FUNCTION_BLOCK T_AdsWrite EXTENDS T_NamedBase IMPLEMENTS I_TaskState;
VAR
   _readWriteOpts : ST_AdsReadWriteOptions;

   write : ADSWRITE;
   {attribute 'to_String'}
   state, prevState : (
      IDLE,
      REQUEST,
      WAIT_FOR_RESPONSE,
      DONE_STATE,
      ERROR_STATE
   );

   lastErrorId : UDINT;

END_VAR
VAR CONSTANT
   NO_ERR : UDINT := 0;
   LOG_DEBUG : DWORD := 0;
   LOG_INFO : DWORD := ADSLOG_MSGTYPE_HINT;
   LOG_WARNING : DWORD := ADSLOG_MSGTYPE_WARN;
   LOG_ERROR : DWORD := ADSLOG_MSGTYPE_ERROR;
END_VAR

CASE state OF

   IDlE:
      IsEntryActionAndLog();

   REQUEST:
      IsEntryActionAndLog();

      lastErrorId := NO_ERR;
      write.WRITE := TRUE;
      state := WAIT_FOR_RESPONSE;

   WAIT_FOR_RESPONSE:
      IsEntryActionAndLog();

      IF write.ERR THEN
         state := ERROR_STATE;

      ELSIF NOT write.BUSY THEN
         state := DONE_STATE;

      END_IF

   DONE_STATE:
      IsEntryActionAndLog();

   ERROR_STATE:
      IF IsEntryActionAndLog() THEN
         lastErrorId := write.ERRID;

      END_IF

END_CASE

write.WRITE R= NOT Busy;
write();

PROPERTY Busy : BOOL
GET
Busy :=
   NOT Done
   AND NOT Error
   AND state <> IDLE;
END_GET
END_PROPERTY

PROPERTY Done : BOOL
GET
Done := state = DONE_STATE;
END_GET
END_PROPERTY

PROPERTY Error : BOOL
GET
Error := state = ERROR_STATE;
END_GET
END_PROPERTY

METHOD PRIVATE IsEntryActionAndLog : BOOL
IsEntryActionAndLog := prevState <> state;

IF NOT IsEntryActionAndLog THEN
   RETURN;
END_IF

LogDebug(
   Msg := F_Concat3(TO_STRING(prevState), ' transition to state ', TO_STRING(state))
);

prevState := state;
END_METHOD

METHOD TryRequest : BOOL
VAR_INPUT
   readWriteOptions : ST_AdsReadWriteOptions;
END_VAR
VAR_OUTPUT
   status : I_TaskState;
END_VAR
VAR CONSTANT
   NO_HANDLE : DWORD := 0;
END_VAR
IF Busy THEN
   LogWarning('Cannot TryRequest as Busy');
   RETURN;

END_IF

_readWriteOpts := readWriteOptions;
write(
   NETID := F_GetAmsNetId(_readWriteOpts.AdsAddress.netId),
   PORT := _readWriteOpts.AdsAddress.port,
   IDXGRP := _readWriteOpts.IndexGroup,
   IDXOFFS := _readWriteOpts.IndexOffset,
   LEN := _readWriteOpts.WriteParams.cbLen,
   SRCADDR := _readWriteOpts.WriteParams.pData,
   TMOUT := _readWriteOpts.Timeout
);

state := REQUEST;

TryRequest := TRUE;
status := THIS^;
END_METHOD

END_FUNCTION_BLOCK

(* stored: Version 1.1.0.1, ProductVersion 3.1.4024.9
   POU T_AdsWrite: Id {74fc4771-e5ab-48d0-b43d-d9873b62fcd2}, SpecialFunc None
   Property Busy: Id {df1e7010-b73f-49a8-b73d-fecf48c237fe}
   Get Get: Id {ce11126a-c87e-4d91-9961-ce674e1ad851}
   Property Done: Id {4b41d635-85a2-44d3-8128-2176e45986fb}
   Get Get: Id {fa3c8a89-c61d-4994-beec-9b5315440b7d}
   Property Error: Id {d9696f66-3622-4c64-a992-5010867801d3}
   Get Get: Id {3c4509eb-058c-45e0-be33-93454c2ff8ec}
   Method IsEntryActionAndLog: Id {c15a70aa-f7c8-4531-add7-9369bbc586d9}
   Method TryRequest: Id {4c4186ee-9a01-46b0-b614-bdcd8a923f22} *)
